// TIA Portal V19 export
ORGANIZATION_BLOCK "A03_OB1"   // OB1, LAD, ProgramCycle
TITLE = "Main Program Sweep (Cycle)"
// stored: SetENOAutomatically false
   VAR_INPUT
      Initial_Call : Bool;   // Initial call of this OB
      Remanence : Bool;   // =True, if remanent data are available
   END_VAR
BEGIN

REGION Network 1
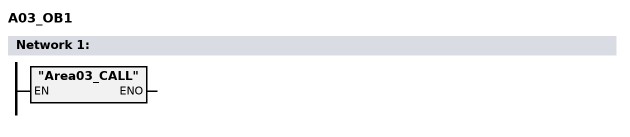
   RUNG wire#powerrail
      "Area03_CALL"()
   END_RUNG
   // the same network as SCL:
   "Area03_CALL"();
END_REGION
END_ORGANIZATION_BLOCK
